Staubli VAL3: buildList.pgx

program buildList()
  local num l_nSize
  local string l_sInstruction
  local num i
  local num j
  local mdesc l_mDesc
  local num l_nTcpAction
  local string l_sEmpty
  local bool false
  local num l_nZero
  local bool l_bToStop
  local TrajectoryItem l_tTraj
begin
  // INIT the list
  l_sEmpty=""
  call use:stringCopy(l_sEmpty,sList)
  // Build the list
  call trajType:getSizeItem(false,l_nSize)
  for i=0 to l_nSize-1
    if bLarge
      // show the instruction
      l_bToStop=false
      l_nZero=0
      call trajType:getTrajItem(l_tTraj,i)
      switch l_tTraj.nTcpAction
        case 1
          l_sInstruction="[ON],"
        break
        case 2
          l_sInstruction="[OFF],"
        break
        default
          l_sInstruction=""
        break
      endSwitch
      // get all the action
      l_sInstruction=l_sInstruction+l_tTraj.iInstr[0].sType+" "+l_tTraj.iInstr[0].sData
      for j=1 to size(l_tTraj.iInstr)-1
        l_sInstruction=l_sInstruction+","+l_tTraj.iInstr[j].sType+" "+l_tTraj.iInstr[j].sData
      endFor
      call use:typeLen(0,12,l_sInstruction,40)
    else
      call trajType:getTrajItem(l_tTraj,i)
      l_sInstruction=l_tTraj.comment
    endIf
    // insert the line
    call listAdd(toString("2",i+1)+" "+l_sInstruction)
  endFor
  // update
  use:bUseRefresh=true
end
